TYPE ST_FeederInProduce :
STRUCT
	CurPos			: LREAL;
	BasePos 		: LREAL;

	StillPos			: LREAL;
	TouchPos		: LREAL;
	TouchFeederIdx	: INT;

END_STRUCT
END_TYPE

(* stored: Version 1.1.0.1, ProductVersion 3.1.4024.9
   DUT ST_FeederInProduce: Id {54f195e3-ec09-406c-a084-0a4dd9b5e5af} *)
